KUKA KRL data list: to_home_R2.dat

&ACCESS RVO1
&COMMENT Przejazd do HOME_POS
&PARAM DISKPATH = KRC:\R1\Program\dodatkowe
DEFDAT to_home_R2 PUBLIC
;FOLD EXTERNAL DECLARATIONS;%{PE}%MKUKATPBASIS,%CEXT,%VCOMMON,%P
;FOLD BASISTECH EXT;%{PE}%MKUKATPBASIS,%CEXT,%VEXT,%P
EXT  BAS (BAS_COMMAND  :IN,REAL  :IN )
DECL INT SUCCESS
;ENDFOLD (BASISTECH EXT)
;FOLD USER EXT;%{E}%MKUKATPUSER,%CEXT,%VEXT,%P
;Make here your modifications

;ENDFOLD (USER EXT)
;ENDFOLD (EXTERNAL DECLERATIONS)

DECL BASIS_SUGG_T LAST_BASIS={POINT1[] "NearHomePos",POINT2[] "NearHomePos",CP_PARAMS[] "CPDAT0",PTP_PARAMS[] "DEFAULT",CONT[] " ",CP_VEL[] "2.0",PTP_VEL[] "10",SYNC_PARAMS[] "SYNCDAT ",SPL_NAME[] "S0 "}
DECL PDAT PPDATH={VEL 100.000,ACC 100.000,APO_DIST 100.000,APO_MODE #CDIS,GEAR_JERK 100.000,EXAX_IGN 0}
DECL MODULEPARAM_T LAST_TP_PARAMS={PARAMS[] "Kuka.MoveDataPtpName=PDATH; Kuka.MovementDataPdat.apo_mode=#CDIS; Kuka.MovementDataPdat.apo_dist=100; Kuka.MovementData.vel=100; Kuka.MovementData.acc=100; Kuka.MovementData.gear_jerk=100; Kuka.MovementData.exax_ign=0; Kuka.VelocityPtp=10; Kuka.BlendingEnabled=False; Kuka.CurrentCDSetIndex=0; Kuka.VelocityFieldEnabled=False; Kuka.ColDetectFieldEnabled=False; Kuka.MovementParameterFieldEnabled=False; Kuka.IsAngleEnabled=False"}

ENDDAT
